// SIMATIC S7-200 project (STEP 7-Micro/WIN), CPU 226 REL 02.01

ORGANIZATION_BLOCK 主程序:OB1
TITLE=这是我做的通过自由口通讯进行温度控制的PLC历程。我用了三种方法实现，这是我想的方法C，供大家一起参考。
// 注释：系统启动时，通过检测首次扫描标志，自动将通讯端口配置设置为特定参数，确保通讯波特率、数据位和停止位与上位机完美匹配，否则通讯将无法正常建立。系统将代表生产参数的预设数据分别写入发送数据缓冲区1、发送数据缓冲区2和发送数据缓冲区3，这些数据必须在发送前准备好且格式正确，以保证上位机能够准确解析。发送字节数被设置为6，确保每次发送的数据长度固定为6个字节，避免因数据长度不匹配导致发送不完整或多余的情况。运行过程中，每当发送触发信号的上升沿到来时，系统通过通讯端口执行发送指令，将发送字节数指定的6个字节数据从指定地址发送到上位机。
// 
BEGIN
Network 1 // 网络标题
// 网络注释
LD     SM0.1
MOVB   16#9, SMB30
MOVW   16#5337, VW100
MOVW   16#2D32, VW102
MOVW   16#3030, VW104
MOVB   6, VB99
?000
Network 2
LD     SM0.5
EU
XMT    VB99, 0
END_ORGANIZATION_BLOCK
